{attribute 'GeneratedUsingTerminal: AMP8000-0030-0103-0103'}
{attribute addProperty BoxType "AMP8000-0030-0103-0103"}
{attribute addProperty Id "FSOEAT %Q*FSOE_BB3344D68"}
{attribute addProperty CRC "1505767614"}
{attribute addProperty Size "8"}
TYPE Standard_Outputdata_59C030BE EXTENDS OutputBase_10CEE7DE :
STRUCT
	{attribute addProperty Name "FSOE"}
	FSOE AT %Q* : FSOE_BB3344D6;
END_STRUCT
END_TYPE

(* stored: Version 1.2.0.0, ProductVersion 3.1.4024.11
   DUT Standard_Outputdata_59C030BE: Id {059d53d1-39bf-4f3f-8653-ed129636a9ab} *)
